GLOBALCONSTANTS DefaultPool_Numeric (* Numeric object pool constants (ID, Scale, Offset, Decimals) *)
  PACKAGE Uebungen::const::UT;
  VAR_GLOBAL CONSTANT
    InputNumber_I1_N : logiBUS::utils::conversion::phys::NumericObjectPool_S := (u16ObjId := 9000, r32Scale := 1.0, i32Offset := 0, u8Decimals := 0);
    InputNumber_I2_N : logiBUS::utils::conversion::phys::NumericObjectPool_S := (u16ObjId := 9001, r32Scale := 1.0, i32Offset := 0, u8Decimals := 0);
    InputNumber_I3_N : logiBUS::utils::conversion::phys::NumericObjectPool_S := (u16ObjId := 9002, r32Scale := 0.01, i32Offset := -100000, u8Decimals := 2);
    InputNumber_I4_N : logiBUS::utils::conversion::phys::NumericObjectPool_S := (u16ObjId := 9003, r32Scale := 0.01, i32Offset := -100000, u8Decimals := 2);
    OutputNumber_N1_N : logiBUS::utils::conversion::phys::NumericObjectPool_S := (u16ObjId := 12000, r32Scale := 1.0, i32Offset := 0, u8Decimals := 0);
    OutputNumber_N2_N : logiBUS::utils::conversion::phys::NumericObjectPool_S := (u16ObjId := 12001, r32Scale := 1.0, i32Offset := 0, u8Decimals := 0);
    OutputNumber_N3_N : logiBUS::utils::conversion::phys::NumericObjectPool_S := (u16ObjId := 12002, r32Scale := 0.01, i32Offset := -100000, u8Decimals := 2);
  END_VAR
END_GLOBALCONSTANTS
